// TIA Portal V17 export
// export: Created 2025-03-07T09:16:29.6462684Z, ExportSetting WithDefaults, DisplayName Totally Integrated Automation Portal, DisplayVersion V17 Update 8, DisplayName TIA Portal Openness, DisplayVersion V17 Update 8, DisplayName TIA Portal Version Control Interface, DisplayVersion V17, DisplayName SINAMICS Startdrive Advanced, DisplayVersion V17 SP2, DisplayName SINAMICS Startdrive G110M, G120, G120C, G120D, G120P, G115D, DisplayVersion V17 SP2, DisplayName SINAMICS Startdrive G130, G150, S120, S150, SINAMICS MV, S210, DisplayVersion V17 SP2, DisplayName STEP 7 Professional, DisplayVersion V17 Update 8, DisplayName SINUMERIK ONE STEP 7 Toolbox, DisplayVersion V17 Update 12, DisplayName SINUMERIK 840D sl STEP 7 Toolbox, DisplayVersion V17 Update 12, DisplayName STEP 7 Safety, DisplayVersion V17 Update 6, DisplayName WinCC Advanced, DisplayVersion V17 Update 8
DATA_BLOCK "LBP_Chan7"   // DB27
TITLE = Channel-specific signals / Señales específicas de canal / Kanalspezifische Signale
{ S7_Optimized_Access := 'FALSE'; DB_Accessible_From_OPC_UA := 'FALSE' }
AUTHOR : SINUMERIK
FAMILY : SINUMERIK_ONE
VERSION : 6.15
// Interface between user program and channel, contains signals from/to channel 7 / La interfaz entre el programa de usuario y el canal contiene señales desde/hacia el canal 7 / Schnittstelle zwischen Anwenderprogramm und Kanal, enthält Signale von/an Kanal 7
// stored: AutoNumber false, DBAccessibleFromOPCUA false, DBAccessibleFromWebserver true, InstanceOfName LBP_typeChanX, InstanceOfType UDT, IsOnlyStoredInLoadMemory false, IsWriteProtectedInAS false
"LBP_typeChanX"
   // VAR RETAIN
   //    f0_0 : Bool;
   //    f0_1 : Bool;
   //    f0_2 : Bool;
   //    A_DRF : Bool;
   //    A_SBL : Bool;
   //    A_M01 : Bool;
   //    A_DRY : Bool;
   //    f0_7 : Bool;
   //    A_Ref : Bool;
   //    A_ProtZone : Bool;
   //    A_SynOff : Bool;
   //    A_TM_TimOut : Bool;
   //    A_CLC_Stop : Bool;
   //    A_CLC_OR : Bool;
   //    A_PLC_ActCompl : Bool;
   //    A_ProgTest : Bool;
   //    A_SKP0 : Bool;
   //    A_SKP1 : Bool;
   //    A_SKP2 : Bool;
   //    A_SKP3 : Bool;
   //    A_SKP4 : Bool;
   //    A_SKP5 : Bool;
   //    A_SKP6 : Bool;
   //    A_SKP7 : Bool;
   //    A_StrokEnab : Bool;
   //    A_ManStrokEnab : Bool;
   //    A_StrokSup : Bool;
   //    A_StrokDelayed : Bool;
   //    A_StrokStop : Bool;
   //    A_ManRelStroke2 : Bool;
   //    A3_6 : Bool;
   //    A3_7 : Bool;
   //    A_FD_OR : Byte;
   //    A_RT_OR : Byte;
   //    A_FDdisable : Bool;
   //    A_RIdisable : Bool;
   //    A_DeleteDTG : Bool;
   //    A_SP_Clear : Bool;
   //    A_ProgAbort : Bool;
   //    A_F_Limit : Bool;
   //    A_RT_ORA : Bool;
   //    A_FD_ORA : Bool;
   //    A_NCStartDisabl : Bool;
   //    A_NCStart : Bool;
   //    A_NCStopBlock : Bool;
   //    A_NCStop : Bool;
   //    A_NCStopASp : Bool;
   //    A_SuppStartLock : Bool;
   //    A_CfgStopFunc : Bool;
   //    A_Reset : Bool;
   //    A_MRP : Array[1..10] of Bool;
   //    A_CSP : Array[1..10] of Bool;
   //    A_Geo : Array[1..3] of Struct
   //       HW1 : Bool;
   //       HW2 : Bool;
   //       HW3 : Bool;
   //       FDStop : Bool;
   //       Disabl : Bool;
   //       RapidTrOR : Bool;
   //       Minus : Bool;
   //       Plus : Bool;
   //       INC1 : Bool;
   //       INC10 : Bool;
   //       INC100 : Bool;
   //       INC1000 : Bool;
   //       INC10000 : Bool;
   //       INCVar : Bool;
   //       ContManTravel : Bool;
   //       f1_7 : Bool;
   //       OEM : Byte;
   //       InvHWDirOfRot : Bool;
   //       f3_1 : Bool;
   //       f3_2 : Bool;
   //       f3_3 : Bool;
   //       f3_4 : Bool;
   //       f3_5 : Bool;
   //       f3_6 : Bool;
   //       f3_7 : Bool;
   //    END_STRUCT;
   //    f24_0 : Bool;
   //    E_MMC_CfgStopFunc : Bool;
   //    f24_2 : Bool;
   //    E_MMC_DRF : Bool;
   //    E_MMC_M01AssocNC : Bool;
   //    E_MMC_M01 : Bool;
   //    E_MMC_DRY : Bool;
   //    f24_7 : Bool;
   //    E_MMC_REPOSPM_0 : Bool;
   //    E_MMC_REPOSPM_1 : Bool;
   //    E_MMC_REPOSPM_2 : Bool;
   //    E_MMC_FD_OR4RT_OR : Bool;
   //    E_MMC_REPOSMode : Bool;
   //    f25_5 : Bool;
   //    f25_6 : Bool;
   //    E_MMC_ProgTest : Bool;
   //    E_MMC_SKP0 : Bool;
   //    E_MMC_SKP1 : Bool;
   //    E_MMC_SKP2 : Bool;
   //    E_MMC_SKP3 : Bool;
   //    E_MMC_SKP4 : Bool;
   //    E_MMC_SKP5 : Bool;
   //    E_MMC_SKP6 : Bool;
   //    E_MMC_SKP7 : Bool;
   //    E_MMC_SKP8 : Bool;
   //    E_MMC_SKP9 : Bool;
   //    f27_2 : Bool;
   //    f27_3 : Bool;
   //    f27_4 : Bool;
   //    f27_5 : Bool;
   //    f27_6 : Bool;
   //    f27_7 : Bool;
   //    A_OEM : Byte;
   //    A_FixedFD1 : Bool;
   //    A_FixedFD2 : Bool;
   //    A_FixedFD3 : Bool;
   //    A_FixedFD4 : Bool;
   //    A_PTP_Travel : Bool;
   //    A_DisablWP_Counter : Bool;
   //    A_DisablWearMon : Bool;
   //    A_DontDisablTool : Bool;
   //    A_ContHW1 : Bool;
   //    A_ContHW2 : Bool;
   //    A_ContHW3 : Bool;
   //    A_ContHWsim : Bool;
   //    A_ContHWneg : Bool;
   //    A_NCKrelatedM01 : Bool;
   //    A_JOG_Circles : Bool;
   //    A_NoToolChangeCmd : Bool;
   //    A_REPOSPM_0 : Bool;
   //    A_REPOSPM_1 : Bool;
   //    A_REPOSPM_2 : Bool;
   //    f31_3 : Bool;
   //    A_REPOSMode : Bool;
   //    A_InvCHWDirOfRot : Bool;
   //    A_SKP8 : Bool;
   //    A_SKP9 : Bool;
   //    E_ExecExtern : Bool;
   //    f32_1 : Bool;
   //    f32_2 : Bool;
   //    E_ActBlock : Bool;
   //    E_BegBlock : Bool;
   //    E_M01 : Bool;
   //    E_LastActBlock : Bool;
   //    f32_7 : Bool;
   //    E_Ref : Bool;
   //    E_OrieToolholder : Bool;
   //    E_RevFD : Bool;
   //    E_HWOverlay : Bool;
   //    E_BlockSearch : Bool;
   //    E_M30 : Bool;
   //    E_Transform : Bool;
   //    E_ProgTest : Bool;
   //    E_OEMChan : Byte;
   //    E_ProgRunning : Bool;
   //    E_ProgWait : Bool;
   //    E_ProgStop : Bool;
   //    E_ProgInterrupt : Bool;
   //    E_ProgAborted : Bool;
   //    E_ChanActive : Bool;
   //    E_ChanInterrupt : Bool;
   //    E_ChanReset : Bool;
   //    E_StartReq : Bool;
   //    E_StopReq : Bool;
   //    E_AxesRef : Bool;
   //    E_AxesStop : Bool;
   //    E_IR_Activ : Bool;
   //    E_ChanRO : Bool;
   //    E_NCKalarmChan : Bool;
   //    E_NCKalarmStop : Bool;
   //    E_CHW1 : Bool;
   //    E_CHW2 : Bool;
   //    E_CHW3 : Bool;
   //    E_CLC : Bool;
   //    E_CLCStopLL : Bool;
   //    E_CLCStopUL : Bool;
   //    E_RIEnabIgnored : Bool;
   //    E_StopBlkEndSBLsuppr : Bool;
   //    E_StrokeEA : Bool;
   //    E_AcknManStrokEnab : Bool;
   //    f38_2 : Bool;
   //    f38_3 : Bool;
   //    f38_4 : Bool;
   //    f38_5 : Bool;
   //    f38_6 : Bool;
   //    f38_7 : Bool;
   //    E_ProtZoneNOK : Bool;
   //    E_NCalarmWithProgStop : Bool;
   //    f39_2 : Bool;
   //    f39_3 : Bool;
   //    E_SblStopAtBlockEnd : Bool;
   //    E_InvCHWDirOfRot : Bool;
   //    E_CfgStopFuncActive : Bool;
   //    E_CfgStopAtBlockEnd : Bool;
   //    E_Geo : Array[1..3] of Struct
   //       HW1 : Bool;
   //       HW2 : Bool;
   //       HW3 : Bool;
   //       f0_3 : Bool;
   //       TReqMinus : Bool;
   //       TReqPlus : Bool;
   //       TCMinus : Bool;
   //       TCPlus : Bool;
   //       INC1 : Bool;
   //       INC10 : Bool;
   //       INC100 : Bool;
   //       INC1000 : Bool;
   //       INC10000 : Bool;
   //       INCVar : Bool;
   //       ContManTravelAct : Bool;
   //       f1_7 : Bool;
   //       OEM : Byte;
   //       InvHWDirOfRot : Bool;
   //       f3_1 : Bool;
   //       f3_2 : Bool;
   //       f3_3 : Bool;
   //       f3_4 : Bool;
   //       f3_5 : Bool;
   //       f3_6 : Bool;
   //       f3_7 : Bool;
   //       f4 : Byte;
   //    END_STRUCT;
   //    M1Change : Bool;
   //    M2Change : Bool;
   //    M3Change : Bool;
   //    M4Change : Bool;
   //    M5Change : Bool;
   //    f58_5 : Bool;
   //    f58_6 : Bool;
   //    f58_7 : Bool;
   //    M1NDec : Bool;
   //    M2NDec : Bool;
   //    M3NDec : Bool;
   //    M4NDec : Bool;
   //    M5NDec : Bool;
   //    f59_5 : Bool;
   //    f59_6 : Bool;
   //    f59_7 : Bool;
   //    S1Change : Bool;
   //    S2Change : Bool;
   //    S3Change : Bool;
   //    f60_3 : Bool;
   //    S1Quick : Bool;
   //    S2Quick : Bool;
   //    S3Quick : Bool;
   //    f60_7 : Bool;
   //    T1Change : Bool;
   //    T2Change : Bool;
   //    T3Change : Bool;
   //    f61_3 : Bool;
   //    T1Quick : Bool;
   //    T2Quick : Bool;
   //    T3Quick : Bool;
   //    f61_7 : Bool;
   //    D1Change : Bool;
   //    D2Change : Bool;
   //    D3Change : Bool;
   //    f62_3 : Bool;
   //    D1Quick : Bool;
   //    D2Quick : Bool;
   //    D3Quick : Bool;
   //    f62_7 : Bool;
   //    EChange : Bool;
   //    f63_1 : Bool;
   //    f63_2 : Bool;
   //    f63_3 : Bool;
   //    EQuick : Bool;
   //    f63_5 : Bool;
   //    f63_6 : Bool;
   //    f63_7 : Bool;
   //    H1Change : Bool;
   //    H2Change : Bool;
   //    H3Change : Bool;
   //    f64_3 : Bool;
   //    H1Quick : Bool;
   //    H2Quick : Bool;
   //    H3Quick : Bool;
   //    f64_7 : Bool;
   //    F1Change : Bool;
   //    F2Change : Bool;
   //    F3Change : Bool;
   //    F4Change : Bool;
   //    F5Change : Bool;
   //    F6Change : Bool;
   //    f65_6 : Bool;
   //    f65_7 : Bool;
   //    M1Quick : Bool;
   //    M2Quick : Bool;
   //    M3Quick : Bool;
   //    M4Quick : Bool;
   //    M5Quick : Bool;
   //    f66_5 : Bool;
   //    f66_6 : Bool;
   //    f66_7 : Bool;
   //    F1Quick : Bool;
   //    F2Quick : Bool;
   //    F3Quick : Bool;
   //    F4Quick : Bool;
   //    F5Quick : Bool;
   //    F6Quick : Bool;
   //    f67_6 : Bool;
   //    f67_7 : Bool;
   //    ExtM1 : Int;
   //    M1 : DInt;
   //    ExtM2 : Int;
   //    M2 : DInt;
   //    ExtM3 : Int;
   //    M3 : DInt;
   //    ExtM4 : Int;
   //    M4 : DInt;
   //    ExtM5 : Int;
   //    M5 : DInt;
   //    ExtS1 : Int;
   //    S1 : Real;
   //    ExtS2 : Int;
   //    S2 : Real;
   //    ExtS3 : Int;
   //    S3 : Real;
   //    ExtT1 : Int;
   //    T1 : Int;
   //    ExtT2 : Int;
   //    T2 : Int;
   //    ExtT3 : Int;
   //    T3 : Int;
   //    ExtD1 : Byte;
   //    D1 : Byte;
   //    ExtD2 : Byte;
   //    D2 : Byte;
   //    ExtD3 : Byte;
   //    D3 : Byte;
   //    ExtE : Int;
   //    "E" : Real;
   //    ExtH1 : Int;
   //    H1 : Real;
   //    ExtH2 : Int;
   //    H2 : Real;
   //    ExtH3 : Int;
   //    H3 : Real;
   //    ExtF1 : Int;
   //    F1 : Real;
   //    ExtF2 : Int;
   //    F2 : Real;
   //    ExtF3 : Int;
   //    F3 : Real;
   //    ExtF4 : Int;
   //    F4 : Real;
   //    ExtF5 : Int;
   //    F5 : Real;
   //    ExtF6 : Int;
   //    F6 : Real;
   //    MDyn : Array[0..99] of Bool;
   //    GAct : Array[1..64] of Byte;
   //    E_MRPactivated : Array[1..10] of Bool;
   //    E_CSPactivated : Array[1..10] of Bool;
   //    E_MRPViolated : Array[1..10] of Bool;
   //    E_CSPViolated : Array[1..10] of Bool;
   //    f_280_0 : Bool;
   //    A_Str_Synon : Bool;
   //    f_280_2 : Bool;
   //    f_280_3 : Bool;
   //    f_280_4 : Bool;
   //    f_280_5 : Bool;
   //    f_280_6 : Bool;
   //    f_280_7 : Bool;
   //    f_281_0 : Bool;
   //    A_Str_Synfrom : Bool;
   //    f_281_2 : Bool;
   //    f_281_3 : Bool;
   //    f_281_4 : Bool;
   //    f_281_5 : Bool;
   //    f_281_6 : Bool;
   //    f_281_7 : Bool;
   //    f_282 : Int;
   //    f_284 : Int;
   //    f_286 : Int;
   //    f_288 : Int;
   //    f_290 : Int;
   //    f_292 : Int;
   //    f_294 : Int;
   //    f_296 : Int;
   //    f_298 : Int;
   //    A_SynDisabl : Array[1..64] of Bool;
   //    E_SynDisabled : Array[1..64] of Bool;
   //    E_G00 : Bool;
   //    f316_1 : Bool;
   //    f316_2 : Bool;
   //    f316_3 : Bool;
   //    f316_4 : Bool;
   //    f316_5 : Bool;
   //    f316_6 : Bool;
   //    f316_7 : Bool;
   //    E_ExtLang : Bool;
   //    E_WS_Setp : Bool;
   //    f317_2 : Bool;
   //    f317_3 : Bool;
   //    f317_4 : Bool;
   //    E_DriveTest : Bool;
   //    E_PTP_Travel : Bool;
   //    E_ToolMissing : Bool;
   //    E_ASUP_Stop : Bool;
   //    E_SearchAct : Bool;
   //    E_TOFF : Bool;
   //    E_TOFFmovem : Bool;
   //    E_StopDelayed : Bool;
   //    E_AssM01 : Bool;
   //    E_DRY : Bool;
   //    E_Overstore : Bool;
   //    E_REPOS_EdgeAckn : Bool;
   //    E_REPOS_PMode0 : Bool;
   //    E_REPOS_PMode1 : Bool;
   //    E_REPOS_PMode2 : Bool;
   //    E_DelayFTS : Bool;
   //    E_REPOS_DEFERRA : Bool;
   //    E_Stop_NoDelayR : Bool;
   //    E_NoToolChangeCmd : Bool;
   //    A_Ori : Array[1..3] of Struct
   //       HW1 : Bool;
   //       HW2 : Bool;
   //       HW3 : Bool;
   //       FDStop : Bool;
   //       Disabl : Bool;
   //       RapidTrOR : Bool;
   //       Minus : Bool;
   //       Plus : Bool;
   //       INC1 : Bool;
   //       INC10 : Bool;
   //       INC100 : Bool;
   //       INC1000 : Bool;
   //       INC10000 : Bool;
   //       INCVar : Bool;
   //       OEM : Byte;
   //       InvHWDirOfRot : Bool;
   //       f3_1 : Bool;
   //       f3_2 : Bool;
   //       f3_3 : Bool;
   //       f3_4 : Bool;
   //       f3_5 : Bool;
   //       f3_6 : Bool;
   //       f3_7 : Bool;
   //    END_STRUCT;
   //    E_Ori : Array[1..3] of Struct
   //       HW1 : Bool;
   //       HW2 : Bool;
   //       HW3 : Bool;
   //       f0_3 : Bool;
   //       TReqMinus : Bool;
   //       TReqPlus : Bool;
   //       TCMinus : Bool;
   //       TCPlus : Bool;
   //       INC1 : Bool;
   //       INC10 : Bool;
   //       INC100 : Bool;
   //       INC1000 : Bool;
   //       INC10000 : Bool;
   //       INCVar : Bool;
   //       OEM : Byte;
   //       InvHWDirOfRot : Bool;
   //       f3_1 : Bool;
   //       f3_2 : Bool;
   //       f3_3 : Bool;
   //       f3_4 : Bool;
   //       f3_5 : Bool;
   //       f3_6 : Bool;
   //       f3_7 : Bool;
   //    END_STRUCT;
   //    E_TPrewarnLimit : Bool;
   //    E_TLimit : Bool;
   //    E_TNewRepl : Bool;
   //    E_TLastRepl : Bool;
   //    f344_4 : Bool;
   //    f344_5 : Bool;
   //    f344_6 : Bool;
   //    f344_7 : Bool;
   //    f345 : Byte;
   //    f346 : Byte;
   //    f347 : Byte;
   //    E_TNoPrewarnLimit : DInt;
   //    E_TNoLimit : DInt;
   //    E_TNoNewRepl : DInt;
   //    E_TNoLastRepl : DInt;
   //    E_Cycle_Sig : Array[0..15] of Bool;
   //    A_Cycle_Sig : Array[0..15] of Bool;
   //    E_OEM_TechnoSig : Array[0..31] of Bool;
   //    A_OEM_TechnoSig : Array[0..31] of Bool;
   //    E_ProgEvent_Start : Bool;
   //    E_ProgEvent_M30 : Bool;
   //    E_ProgEvent_Reset : Bool;
   //    E_ProgEvent_PowerOn : Bool;
   //    E_ProgEvent_SearchRun : Bool;
   //    f376_5 : Bool;
   //    f376_6 : Bool;
   //    f376_7 : Bool;
   //    E_CollCheckStop : Bool;
   //    E_StopCondition : Bool;
   //    f377_2 : Bool;
   //    f377_3 : Bool;
   //    E_JogRetract : Bool;
   //    E_RetractData : Bool;
   //    E_JOG_Circles : Bool;
   //    f377_7 : Bool;
   //    E_AnyAsup : Bool;
   //    E_SilentAsup : Bool;
   //    f378_2 : Bool;
   //    f378_3 : Bool;
   //    f378_4 : Bool;
   //    f378_5 : Bool;
   //    f378_6 : Bool;
   //    f378_7 : Bool;
   //    f379 : Byte;
   //    f380 : Array[0..31] of Bool;
   //    A_ProgJump : Bool;
   //    f384_1 : Bool;
   //    f384_2 : Bool;
   //    f384_3 : Bool;
   //    f384_4 : Bool;
   //    f384_5 : Bool;
   //    f384_6 : Bool;
   //    f384_7 : Bool;
   //    A_InKeyG1 : Bool;
   //    A_InKeyG2 : Bool;
   //    A_InKeyG3 : Bool;
   //    A_InKeyG4 : Bool;
   //    A_InKeyG5 : Bool;
   //    A_InKeyG6 : Bool;
   //    A_InKeyG7 : Bool;
   //    A_InKeyG8 : Bool;
   //    A_InKeyGEn1 : Bool;
   //    A_InKeyGEn2 : Bool;
   //    A_InKeyGEn3 : Bool;
   //    A_InKeyGEn4 : Bool;
   //    A_InKeyGEn5 : Bool;
   //    A_InKeyGEn6 : Bool;
   //    A_InKeyGEn7 : Bool;
   //    A_InKeyGEn8 : Bool;
   //    A_InKeyGRunIn1 : Bool;
   //    A_InKeyGRunIn2 : Bool;
   //    A_InKeyGRunIn3 : Bool;
   //    A_InKeyGRunIn4 : Bool;
   //    A_InKeyGRunIn5 : Bool;
   //    A_InKeyGRunIn6 : Bool;
   //    A_InKeyGRunIn7 : Bool;
   //    A_InKeyGRunIn8 : Bool;
   //    E_TransformNo : Byte;
   //    f389 : Byte;
   //    E_InKeyGIsEn1 : Bool;
   //    E_InKeyGIsEn2 : Bool;
   //    E_InKeyGIsEn3 : Bool;
   //    E_InKeyGIsEn4 : Bool;
   //    E_InKeyGIsEn5 : Bool;
   //    E_InKeyGIsEn6 : Bool;
   //    E_InKeyGIsEn7 : Bool;
   //    E_InKeyGIsEn8 : Bool;
   //    E_InKeyGRunOut1 : Bool;
   //    E_InKeyGRunOut2 : Bool;
   //    E_InKeyGRunOut3 : Bool;
   //    E_InKeyGRunOut4 : Bool;
   //    E_InKeyGRunOut5 : Bool;
   //    E_InKeyGRunOut6 : Bool;
   //    E_InKeyGRunOut7 : Bool;
   //    E_InKeyGRunOut8 : Bool;
   //    E_CART_JOG_MODE : Byte;
   //    f393 : Byte;
   //    f394 : Byte;
   //    f395 : Byte;
   //    H1_DInt : DInt;
   //    H2_DInt : DInt;
   //    H3_DInt : DInt;
   //    E_AxisSelType : Byte;
   //    E_AxisSelAxis : Byte;
   //    E_AxisSelRequest : Bool;
   //    f410_1 : Bool;
   //    f410_2 : Bool;
   //    f410_3 : Bool;
   //    f410_4 : Bool;
   //    f410_5 : Bool;
   //    f410_6 : Bool;
   //    f410_7 : Bool;
   //    f411 : Byte;
   //    A_AxisSelTypeActive : Byte;
   //    A_AxisSelAxisActive : Byte;
   // END_VAR
BEGIN
END_DATA_BLOCK
